PROGRAM PRG_HallRoom
VAR
	fbLamp : ARRAY[0..3] OF FB_Lamp;
	fbDimmer : ARRAY[0..3] OF FB_Dimmer;
	fbFan: FB_Fan;
	fbCurtain: FB_Curtain;
	i: INT;	
END_VAR


	FOR i := 0 TO 3 BY 1 DO
		fbLamp[i]();
		fbDimmer[i]();
	END_FOR
	fbFan();
	
	fbCurtain();

END_PROGRAM

(* stored: Version 1.1.0.1, ProductVersion 3.1.4024.12
   POU PRG_HallRoom: Id {41486ad6-cc2d-41a2-8753-92a7daf9a437}, SpecialFunc None *)
